(* Logix 5000 project; controller TestController vendor 1 type 14 code 166 rev 32.11; software revision 32.02 *)
// This is a test project

TASK Continuous (continuous, watchdog 500 ms) : MainProgram   // Test continuous task
TASK EventTask (event, rate 10 ms, priority 10, watchdog 500 ms) : EventProgram01   // TestEvent Task
TASK TestTask (periodic, rate 10 ms, priority 10, watchdog 500 ms) : EquipmentPhaseProgram

MODULES
   Local : vendor 1 type 14 code 166 (ICP 0, rev 32.11)
END_MODULES

TYPE AlarmType :   // This is a test alarm type
STRUCT
   DigitalMember : CAM;   // Test digital member
END_STRUCT
END_TYPE

TYPE BoolTest :   // This is a test
STRUCT
   Member01 : BOOL;
   Member02 : BOOL;
   Member04 : BOOL;
   Member05 : BOOL;
END_STRUCT
END_TYPE

TYPE MyStringType :   // This is a test string type
STRUCT
   LEN : DINT;
   DATA : SINT[100];
END_STRUCT
END_TYPE

VAR_GLOBAL   (* controller tags *)
   EquipmentPhaseProgram : PHASE;
   SimpleBool : BOOL; {access None}
   SimpleDint : DINT; {access None}
   SimpleLint : LINT; {access None}
   SimpleSint : SINT; {access None}
        .0   // This is a test
   TestAlarmTag : ALARM; {access None}
   TestAnalogAlarm : ALARM_ANALOG;
   TestArrayTypeTag : ArrayType; {access None}
   TestComplexTag : ComplexType; {access None}
   TestDigitalAlarm : ALARM_DIGITAL;
   TestStringTag : MyStringType; {access None}
   TestTag01 : SimpleType := (IntMember := 14, DintMember := 3); {access Read Only}
END_VAR

PROGRAM EquipmentPhaseProgram
// Test

ROUTINE Resetting   (* ladder *)
END_ROUTINE

ROUTINE Running   (* ladder *)
END_ROUTINE
END_PROGRAM

PROGRAM EventProgram01
END_PROGRAM

PROGRAM MainProgram
END_PROGRAM
